// TwinCAT 3 PLC project Untitled1
// ProgramVersion: 3.1.4023.0
// libraries:
//   ESO LDC Comm Common Library, * (ESO)
//   ESO LDC Motor Library, * (ESO)
//   Tc2_Standard, * (Beckhoff Automation GmbH)
//   Tc2_System, * (Beckhoff Automation GmbH)
//   Tc3_Module, * (Beckhoff Automation GmbH)
//   VisuDialogs, * (System)
//   VisuSymbols,3.5.10.0,System
// project tree:
//   DUTs/ States.TcDUT
//   / GlobalTextList.TcGTLO, PlcTask.TcTTO, Visualization Manager.TcVMO (not stored)
//   POUs/ MAIN.TcPOU
//   VISUs/ Visualization.TcVIS
// real-time tasks:
//   TASK PlcTask: cycle T#10ms, priority 20, ADS port 350
// motion (NC):
//   TASK NC-Task 1 SAF: cycle T#2ms, priority 4, ADS port 501
//   TASK NC-Task 1 SVB: cycle T#10ms, priority 8, ADS port 511
//   AXIS Axis 1 (id 1)
//     OtherSettings: AllowMotionCmdToSlave=true
//     encoder EncType=1
//     drive DrvType=5
//       Analog: TorqueSetpointScale=10, ScaleFactorActTorque=0.1
//       TimeComp: TaskDelayCycles=1
//     controller CtrType=1
//       CtrPara: PriorControlFactor=1
//         Observer: BandWidth=20
//   AXIS Axis 2 (id 2)
//     OtherSettings: AllowMotionCmdToSlave=true
//     encoder EncType=1
//     drive DrvType=5
//       Analog: TorqueSetpointScale=10, ScaleFactorActTorque=0.1
//       TimeComp: TaskDelayCycles=1
//     controller CtrType=1
//       CtrPara: PriorControlFactor=1
//         Observer: BandWidth=20
//   AXIS Axis 3 (id 3)
//     OtherSettings: AllowMotionCmdToSlave=true
//     encoder EncType=1
//     drive DrvType=5
//       Analog: TorqueSetpointScale=10, ScaleFactorActTorque=0.1
//       TimeComp: TaskDelayCycles=1
//     controller CtrType=1
//       CtrPara: PriorControlFactor=1
//         Observer: BandWidth=20
//   AXIS Axis 4 (id 4)
//     OtherSettings: AllowMotionCmdToSlave=true
//     encoder EncType=1
//     drive DrvType=5
//       Analog: TorqueSetpointScale=10, ScaleFactorActTorque=0.1
//       TimeComp: TaskDelayCycles=1
//     controller CtrType=1
//       CtrPara: PriorControlFactor=1
//         Observer: BandWidth=20
// variable links:
//   Untitled1/Untitled1 Instance <-> NC-Task 1 SAF/Axes/Axis 1
//     PlcTask Inputs/MAIN.Motor[1].Axis.NcToPlc <-> Outputs/ToPlc
//     PlcTask Outputs/MAIN.Motor[1].Axis.PlcToNc <-> Inputs/FromPlc
//   Untitled1/Untitled1 Instance <-> NC-Task 1 SAF/Axes/Axis 2
//     PlcTask Inputs/MAIN.Motor[2].Axis.NcToPlc <-> Outputs/ToPlc
//     PlcTask Outputs/MAIN.Motor[2].Axis.PlcToNc <-> Inputs/FromPlc
//   Untitled1/Untitled1 Instance <-> NC-Task 1 SAF/Axes/Axis 3
//     PlcTask Inputs/MAIN.Motor[3].Axis.NcToPlc <-> Outputs/ToPlc
//     PlcTask Outputs/MAIN.Motor[3].Axis.PlcToNc <-> Inputs/FromPlc
//   Untitled1/Untitled1 Instance <-> NC-Task 1 SAF/Axes/Axis 4
//     PlcTask Inputs/MAIN.Motor[4].Axis.NcToPlc <-> Outputs/ToPlc
//     PlcTask Outputs/MAIN.Motor[4].Axis.PlcToNc <-> Inputs/FromPlc
//   Untitled1/Untitled1 Instance <-> Untitled1/Untitled1 Instance
//     PlcTask Inputs/MAIN.Motor[{1..4}].i_bBrake_Stat <-> PlcTask Outputs/MAIN.Simu[{1..4}].q_bBrake_Stat  (4 links)
//     PlcTask Inputs/MAIN.Motor[{1..4}].i_nCouplerState <-> PlcTask Outputs/MAIN.Simu[{1..4}].q_nCouplerState  (4 links)
//     PlcTask Inputs/MAIN.Motor[{1..4}].switches <-> PlcTask Outputs/MAIN.Simu[{1..4}].switches  (4 links)
//     PlcTask Inputs/MAIN.Simu[{1..4}].i_bBrake_Ctrl <-> PlcTask Outputs/MAIN.Motor[{1..4}].q_bBrake_Ctrl  (4 links)

CONFIGURATION Untitled1
    RESOURCE PLC ON TwinCAT3
        TASK PlcTask(INTERVAL := T#10ms, PRIORITY := 20);
        PROGRAM MAIN WITH PlcTask : MAIN;
    END_RESOURCE
END_CONFIGURATION

// ---- DUTs/States.TcDUT
{attribute 'qualified_only'}
{attribute 'strict'}
TYPE States :
(
	Reset := 0,
	Init,
	Enable,
	bLocal,
	MoveType,
	Error,
	Absolute,
	Relative,
	Velocity,
	Stop
);
END_TYPE

// ---- POUs/MAIN.TcPOU
PROGRAM MAIN
VAR
	Motor 					: ARRAY [1..4] OF FB_MOTOR;
	Simu 					: ARRAY [1..4] OF FB_SIM_MOTOR;
	sNames 					: ARRAY [1..4] OF STRING;
	State 					: ARRAY [1..4] OF States;
	previousState 			: ARRAY [1..4] OF States;
	bReset 			AT %I*	: ARRAY [1..4] OF BOOL;
	sMessage 		AT %I*	: ARRAY [1..4] OF STRING;
	bMove 			AT %I*	: ARRAY [1..4] OF BOOL;
	sMovType 		AT %I*	: ARRAY [1..4] OF STRING;
	lrPosition 		AT %I*	: ARRAY [1..4] OF LREAL;
	lrVelocity 		AT %I*	: ARRAY [1..4] OF LREAL;
	
	index					: INT;
	iNumber 				: INT;

	a: INT :=1;
	bStop: ARRAY [1..4] OF BOOL;
END_VAR

// Iniciamos los motores y sus simuladores
FOR index:=1 TO 4 DO
	sNames[index] := CONCAT('Motor', INT_TO_STRING(index));
	Motor[index](sName:=sNames[index], nNOVRAM_DevId:=0);
	Simu[index](ptrCfg:=ADR(Motor[index].cfg), ptrStat:=ADR(Motor[index].stat));
END_FOR

FOR iNumber := 1 TO 4 DO
	ACT_Mot();
END_FOR

//iNumber := 1;
//ACT_Mot();

ACTION ACT_Mot:
// Debido a que este código se basa en comandos RPC debemos poder parar su ejecución en cualquier momento
// si se activa el modo de control local
IF Motor[iNumber].stat.bLocal THEN
	previousState[iNumber] := State[iNumber];
	State[iNumber] := States.bLocal;
END_IF

IF bReset[iNumber] THEN
	State[iNumber] := States.Reset;
END_IF

CASE State[iNumber] OF
	
	States.bLocal :
		// Esperamos hasta que se desactiva el control local y volvemos al estado en el que nos encontrábamos.
		IF NOT Motor[iNumber].stat.bLocal THEN
			State[iNumber] := previousState[iNumber];
		END_IF
	
	States.Error :
		// En caso de error imprimimos el error en pantalla y esperamos a que el usuario nos de el OK para hacer un reset
		sMessage[iNumber] := CONCAT('Motor error: ', Motor[iNumber].stat.sErrorText);
		IF bReset[iNumber] THEN
			State[iNumber] := States.Reset;
		END_IF
		
	States.Stop :
		// En caso de solicitud de stop paramos el motor y volvemos al estado de espera de movimiento
		Motor[iNumber].RPC_Stop();
		State[iNumber] := States.MoveType;
		
	States.Reset :
		// Hacemos el reset y pasamos al estado de init
		Motor[iNumber].RPC_Reset();
		State[iNumber] := States.Init;
		bReset[iNumber] := FALSE;
	
	States.Init :
		// Ejecutamos el init y pasamos al estado de enable
		Motor[iNumber].RPC_Init();
		State[iNumber] := States.Enable;
		
	States.Enable :
		// Esperamos a que acabe la inicialización para realizar el enamble y pasar al siguiente estado
		IF Motor[iNumber].stat.bInitialised THEN
			Motor[iNumber].RPC_Enable();
			State[iNumber] := States.MoveType;
		// En caso de error durante el init pasamos al estado de reset
		ELSIF Motor[iNumber].stat.nStatus = E_MOTOR_STATUS.ERROR THEN
			State[iNumber] := States.Error;
		END_IF
		
	States.MoveType :
		// Comprobamos que no se haya producido ningún error en el movimiento anterior
		IF Motor[iNumber].stat.nStatus = E_MOTOR_STATUS.ERROR THEN
			State[iNumber] := States.Error;
		ELSE
			IF bStop[iNumber] THEN
				State[iNumber] := States.Stop;
				bStop[iNumber] := FALSE;
			// Esperamos a que el usuario active el movimiento para leer qué tipo de movimiento quiere hacer
			ELSIF bMove[iNumber] THEN
				bMove[iNumber] := FALSE;
				IF sMovType[iNumber] = 'Abs' THEN
					State[inumber] := States.Absolute;
					sMessage[iNumber] := '';             // En caso de que hubiese algún mensaje de tipo de movimiento erróneo anterior lo reseteamos
				ELSIF sMovType[iNumber] = 'Rel' THEN
					State[inumber] := States.Relative;
					sMessage[iNumber] := '';
				ELSIF sMovType[iNumber] = 'Vel' THEN
					State[inumber] := States.Velocity;
					sMessage[iNumber] := '';
				ELSE 
					sMessage[iNumber] := 'Wrong movement type input';
				END_IF
			END_IF
		END_IF
		
	States.Absolute :
		// Ejecutamos el movimiento absoluto
		Motor[iNumber].RPC_MoveAbs(in_lrPos := lrPosition[iNumber], in_lrVel := lrVelocity[iNumber]);
		State[iNumber] := States.MoveType;
		
	States.Relative :
		// Ejecutamos el movimiento relativo
		Motor[iNumber].RPC_MoveRel(in_lrPos := lrPosition[iNumber], in_lrVel := lrVelocity[iNumber]);
		State[iNumber] := States.MoveType;
		
	States.Velocity :
		// Ejecutamos el movimiento en velocidad
		Motor[iNumber].RPC_MoveVel(in_lrVel := lrVelocity[iNumber]);
		State[iNumber] := States.MoveType;
		
END_CASE
END_ACTION

END_PROGRAM

// ---- GlobalTextList.TcGTLO
TEXTLIST GlobalTextList
  321 = '%.2d'
  444 = '%.2f'
  537 = '%s'
  714 = 'ACT. POSITION'
  717 = 'ACT. VELOCITY'
  411 = 'Degrees'
  229 = 'Init 1 OK'
  445 = 'Init 2 OK'
  756 = 'Init 3 OK'
  496 = 'Init 4 OK'
  840 = 'MOTOR 1'
  434 = 'MOTOR 2'
  672 = 'MOTOR 3'
  143 = 'MOTOR 4'
  137 = 'MOV. TYPE'
  475 = 'MOVE 1'
  764 = 'MOVE 2'
  204 = 'MOVE 3'
  159 = 'MOVE 4'
  235 = 'POSITION'
  88 = 'Reset 1'
  183 = 'Reset 2'
  225 = 'Reset 3'
  944 = 'Reset 4'
  24 = "Select 'Abs', 'Rel' or 'Vel'"
  152 = 'SET MOV. TYPE'
  105 = 'SET POSITION'
  430 = 'SET VELOCITY'
  922 = 'Stop 1'
  536 = 'Stop 2'
  68 = 'Stop 3'
  323 = 'Stop 4'
  171 = 'VELOCITY'
END_TEXTLIST

// ---- VISUs/Visualization.TcVIS
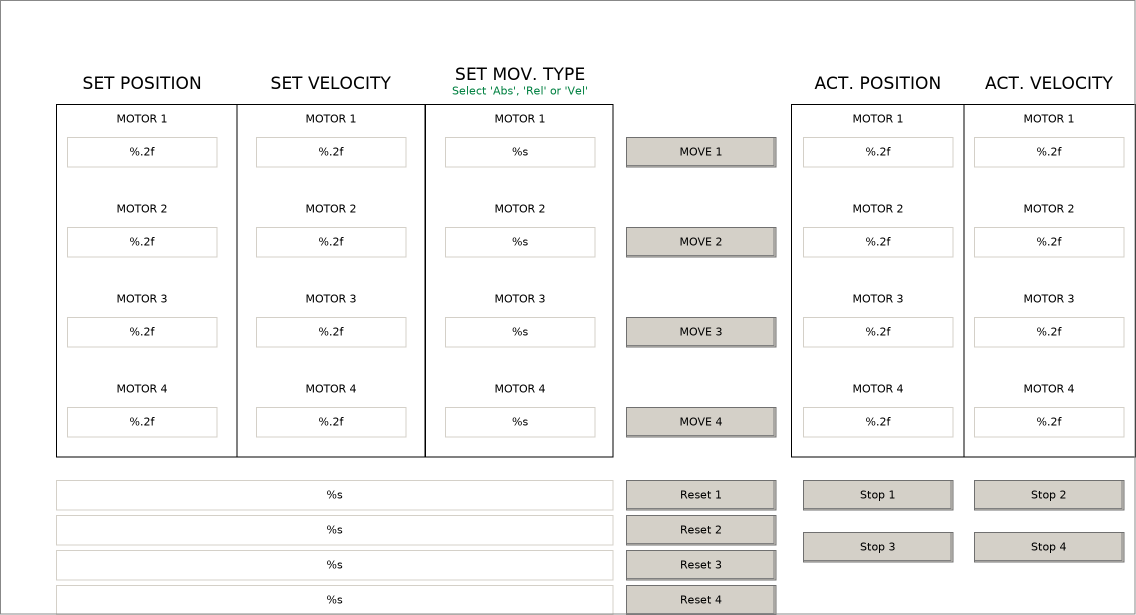
VISUALIZATION Visualization  // 1136x615
    Rectangle (425,104 188x353)
    Rectangle (233,104 192x353)
    Rectangle (56,104 181x353)
    Textfield (67,137 150x30), "%.2f", text variable: MAIN.lrPosition[1]
        OnMouseClick: write the text variable via Default
    Label (67,104 150x30), "MOTOR 1"
    Textfield (67,227 150x30), "%.2f", text variable: MAIN.lrPosition[2]
        OnMouseClick: write the text variable via Default
    Label (67,194 150x30), "MOTOR 2"
    Textfield (67,317 150x30), "%.2f", text variable: MAIN.lrPosition[3]
        OnMouseClick: write the text variable via Default
    Label (67,284 150x30), "MOTOR 3"
    Textfield (67,407 150x30), "%.2f", text variable: MAIN.lrPosition[4]
        OnMouseClick: write the text variable via Default
    Label (67,374 150x30), "MOTOR 4"
    Textfield (256,137 150x30), "%.2f", text variable: MAIN.lrVelocity[1]
        OnMouseClick: write the text variable via Default
    Label (256,104 150x30), "MOTOR 1"
    Textfield (256,227 150x30), "%.2f", text variable: MAIN.lrVelocity[2]
        OnMouseClick: write the text variable via Default
    Label (256,194 150x30), "MOTOR 2"
    Textfield (256,317 150x30), "%.2f", text variable: MAIN.lrVelocity[3]
        OnMouseClick: write the text variable via Default
    Label (256,284 150x30), "MOTOR 3"
    Textfield (256,407 150x30), "%.2f", text variable: MAIN.lrVelocity[4]
        OnMouseClick: write the text variable via Default
    Label (256,374 150x30), "MOTOR 4"
    Textfield (445,137 150x30), "%s", text variable: MAIN.sMovType[1]
        OnMouseClick: write the text variable via Default
    Label (445,104 150x30), "MOTOR 1"
    Textfield (445,227 150x30), "%s", text variable: MAIN.sMovType[2]
        OnMouseClick: write the text variable via Default
    Label (445,194 150x30), "MOTOR 2"
    Textfield (445,317 150x30), "%s", text variable: MAIN.sMovType[3]
        OnMouseClick: write the text variable via Default
    Label (445,284 150x30), "MOTOR 3"
    Textfield (445,407 150x30), "%s", text variable: MAIN.sMovType[4]
        OnMouseClick: write the text variable via Default
    Label (445,374 150x30), "MOTOR 4"
    Label (67,68 150x30), "SET POSITION"
    Label (256,68 150x30), "SET VELOCITY"
    Label (445,59 150x30), "SET MOV. TYPE"
    Rectangle (963,104 173x353)
    Rectangle (791,104 173x353)
    Textfield (803,137 150x30), "%.2f", text variable: MAIN.Motor[1].stat.lrPosActual
    Label (803,104 150x30), "MOTOR 1"
    Textfield (803,227 150x30), "%.2f", text variable: MAIN.Motor[2].stat.lrPosActual
    Label (803,194 150x30), "MOTOR 2"
    Textfield (803,317 150x30), "%.2f", text variable: MAIN.Motor[3].stat.lrPosActual
    Label (803,284 150x30), "MOTOR 3"
    Textfield (803,407 150x30), "%.2f", text variable: MAIN.Motor[4].stat.lrPosActual
    Label (803,374 150x30), "MOTOR 4"
    Textfield (974,137 150x30), "%.2f", text variable: MAIN.Motor[1].stat.lrVelActual
    Label (974,104 150x30), "MOTOR 1"
    Textfield (974,227 150x30), "%.2f", text variable: MAIN.Motor[2].stat.lrVelActual
    Label (974,194 150x30), "MOTOR 2"
    Textfield (974,317 150x30), "%.2f", text variable: MAIN.Motor[3].stat.lrVelActual
    Label (974,284 150x30), "MOTOR 3"
    Textfield (974,407 150x30), "%.2f", text variable: MAIN.Motor[4].stat.lrVelActual
    Label (974,374 150x30), "MOTOR 4"
    Label (803,68 150x30), "ACT. POSITION"
    Label (974,68 150x30), "ACT. VELOCITY"
    Button (626,137 150x30), "MOVE 1"
        tap MAIN.bMove[1] p1329445385=TRUE
    Button (626,227 150x30), "MOVE 2"
        tap MAIN.bMove[2]
    Button (626,317 150x30), "MOVE 3"
        tap MAIN.bMove[3]
    Button (626,407 150x30), "MOVE 4"
        tap MAIN.bMove[4]
    Textfield (56,480 557x30), "%s", text variable: MAIN.sMessage[1]
    Textfield (56,515 557x30), "%s", text variable: MAIN.sMessage[2]
    Textfield (56,550 557x30), "%s", text variable: MAIN.sMessage[3]
    Textfield (56,585 557x30), "%s", text variable: MAIN.sMessage[4]
    Button (626,480 150x30), "Reset 1"
        tap MAIN.bReset[1] p1329445385=TRUE
    Button (626,515 150x30), "Reset 2"
        tap MAIN.bReset[2] p1329445385=TRUE
    Button (626,550 150x30), "Reset 3"
        tap MAIN.bReset[3] p1329445385=TRUE
    Button (626,585 150x30), "Reset 4"
        tap MAIN.bReset[4] p1329445385=TRUE
    Label (445,76 150x30), "Select 'Abs', 'Rel' or 'Vel'"
    Button (803,480 150x30), "Stop 1"
        tap MAIN.bStop[1] p1329445385=TRUE
    Button (974,480 150x30), "Stop 2"
        tap MAIN.bStop[2] p1329445385=TRUE
    Button (803,532 150x30), "Stop 3"
        tap MAIN.bStop[3] p1329445385=TRUE
    Button (974,532 150x30), "Stop 4"
        tap MAIN.bStop[4] p1329445385=TRUE
END_VISUALIZATION
